	(* Internal method *)
	{attribute 'hide'}
	METHOD FB_init : BOOL
	VAR_INPUT
		(*  if TRUE, the retain variables are initialized (warm start / cold start) *)
		bInitRetains : BOOL;
		(*  if TRUE, the instance afterwards gets moved into the copy code (online change) *)
		bInCopyCode : BOOL;
	END_VAR
END_METHOD


	(* Internal method *)
	{attribute 'hide'}
	METHOD FB_exit : BOOL
	VAR_INPUT
		(*  if TRUE, the exit method is called for exiting an instance that is copied afterwards (online change). *)
		bInCopyCode : BOOL;
	END_VAR
END_METHOD


	(* Set the rotation angle in degrees [Â°]. *)
	METHOD SetAngle
	VAR_INPUT
		(* Rotation angle to set in degrees [Â°]. *)
		angle : LREAL;
	END_VAR
END_METHOD


	(* Set the components of this vector to '0.0'. *)
	METHOD SetZero
END_METHOD


	(* Set the components of this orientation. *)
	METHOD SetValues
	VAR_IN_OUT
		(* The position values to set. *)
 {attribute 'GUID' := '340DBC88-CE7F-36B9-693C-9000EEF35F3F'}
				orientation2D : Orientation2D;
	END_VAR
END_METHOD


	(* Get the direction of the local x-axis. *)
	METHOD GetDirectionX
	VAR_IN_OUT
		(* The local x-direction of this orientation. *)
 {attribute 'GUID' := 'FE5FBEA1-CCA0-3BC6-7207-1BBF2A5405AC'}
				localX : TangentXY;
	END_VAR
END_METHOD


	(* Get the direction of the local y-axis. *)
	METHOD GetDirectionY
	VAR_IN_OUT
		(* The local y-direction of this orientation. *)
 {attribute 'GUID' := 'FE5FBEA1-CCA0-3BC6-7207-1BBF2A5405AC'}
				localY : TangentXY;
	END_VAR
END_METHOD


	(* Invert this position. *)
	METHOD Invert
END_METHOD


	(* Multiply an orientation to this orientation. *)
	METHOD ConcatenateWith
	VAR_IN_OUT
		(* Orientation to concatenate with. *)
 {attribute 'GUID' := '340DBC88-CE7F-36B9-693C-9000EEF35F3F'}
				orientation2D : Orientation2D;
	END_VAR
END_METHOD


	(* Turn the orientation. *)
	METHOD TurnByC
	VAR_INPUT
		(* Rotation angle to turn by in degrees [Â°]. *)
		angle : LREAL;
	END_VAR
END_METHOD


	(* Rotate a PositionXY according to this orientation. *)
	METHOD Transform
	VAR_IN_OUT
		(* The orientation to multipy by. *)
 {attribute 'GUID' := '4E15B754-A8FD-31E0-757D-498AD44094D3'}
				positionXY : PositionXY;
	END_VAR
END_METHOD


	PROPERTY angle : LREAL
GET
END_GET
SET
END_SET
END_PROPERTY

END_FUNCTION_BLOCK

// POUs/Spatial/Functions/ConcatenateABC

	{attribute 'TcIecLibraryType'}
	{attribute 'external_name' := 'ConcatenateABC_GUID_C08B4073_E8F0_3BDB_7D4F_B552CCE66755'}
	(* Concatenate two instances of Orientation3D. *)
	FUNCTION ConcatenateABC : BOOL
	VAR_IN_OUT
		rotation0	:	Orientation3D;	(* 1st input orientation of the concatenation. *)
		rotation1	:	Orientation3D;	(* 2nd input orientation of the concatenation. *)
		concatenation	:	Orientation3D;	(* The concatenation of the two input instances. *)
	END_VAR

END_FUNCTION

// POUs/Spatial/Positions/Orientation3D

	{attribute 'c++_compatible'}
	{attribute 'external_name' := 'Orientation3D_GUID_50C17DBD_EDDF_3FDB_7A52_07B790BA3FF3'}
	{attribute 'TcIecLibraryType'}
	{attribute 'no_explicit_call' :='do not call this POU directly'}
	{attribute 'no_assign'}
	(* 3D orientation. All angles in degrees [Â°]. *)
	FUNCTION_BLOCK Orientation3D
	VAR
		(* Rotation around the 1st local axis in degrees [Â°]. *)
		p0 : LREAL;
		(* Rotation around 2nd local axis in degrees [Â°]. *)
		p1 : LREAL;
		(* Rotation around 3rd local axis in degrees [Â°]. *)
		p2 : LREAL;
		(* Defines the rotation order (rotate around local axes from left to right) *)
		 {attribute 'GUID' := 'BF8BCC1E-925E-4A57-801C-CC42AFDDA86D'}
		coordinates : E_RotationCoordinates := E_RotationCoordinates.CBA;
		 {attribute 'hide'}
		_reserved1 : ARRAY [1..84] OF USINT;
	END_VAR


	(* Internal method *)
	{attribute 'hide'}
	METHOD FB_init : BOOL
	VAR_INPUT
		(*  if TRUE, the retain variables are initialized (warm start / cold start) *)
		bInitRetains : BOOL;
		(*  if TRUE, the instance afterwards gets moved into the copy code (online change) *)
		bInCopyCode : BOOL;
	END_VAR
END_METHOD


	(* Internal method *)
	{attribute 'hide'}
	METHOD FB_exit : BOOL
	VAR_INPUT
		(*  if TRUE, the exit method is called for exiting an instance that is copied afterwards (online change). *)
		bInCopyCode : BOOL;
	END_VAR
END_METHOD


	(* Set the components of this vector to '0.0'. *)
	METHOD SetZero
END_METHOD


	(* Set the components of this position. *)
	METHOD SetValues
	VAR_IN_OUT
		(* The position values to set. *)
 {attribute 'GUID' := '50C17DBD-EDDF-3FDB-7A52-07B790BA3FF3'}
				orientation3D : Orientation3D;
	END_VAR
END_METHOD


	(* Set the coordinates of the orientation. *)
	METHOD SetValuesABC
	VAR_INPUT
		(* 1st rotation angle in degrees [Â°]. *)
		phi0 : LREAL;
		(* 2nd rotation angle in degrees [Â°]. *)
		phi1 : LREAL;
		(* 3rd rotation angle in degrees [Â°]. *)
		phi2 : LREAL;
	END_VAR
END_METHOD


	(* Set the coordinates of the orientation. *)
	METHOD SetValuesACB
	VAR_INPUT
		(* 1st rotation angle in degrees [Â°]. *)
		phi0 : LREAL;
		(* 2nd rotation angle in degrees [Â°]. *)
		phi1 : LREAL;
		(* 3rd rotation angle in degrees [Â°]. *)
		phi2 : LREAL;
	END_VAR
END_METHOD


	(* Set the coordinates of the orientation. *)
	METHOD SetValuesBCA
	VAR_INPUT
		(* 1st rotation angle in degrees [Â°]. *)
		phi0 : LREAL;
		(* 2nd rotation angle in degrees [Â°]. *)
		phi1 : LREAL;
		(* 3rd rotation angle in degrees [Â°]. *)
		phi2 : LREAL;
	END_VAR
END_METHOD


	(* Set the coordinates of the orientation. *)
	METHOD SetValuesBAC
	VAR_INPUT
		(* 1st rotation angle in degrees [Â°]. *)
		phi0 : LREAL;
		(* 2nd rotation angle in degrees [Â°]. *)
		phi1 : LREAL;
		(* 3rd rotation angle in degrees [Â°]. *)
		phi2 : LREAL;
	END_VAR
END_METHOD


	(* Set the coordinates of the orientation. *)
	METHOD SetValuesCAB
	VAR_INPUT
		(* 1st rotation angle in degrees [Â°]. *)
		phi0 : LREAL;
		(* 2nd rotation angle in degrees [Â°]. *)
		phi1 : LREAL;
		(* 3rd rotation angle in degrees [Â°]. *)
		phi2 : LREAL;
	END_VAR
END_METHOD


	(* Set the coordinates of the orientation. *)
	METHOD SetValuesCBA
	VAR_INPUT
		(* 1st rotation angle in degrees [Â°]. *)
		phi0 : LREAL;
		(* 2nd rotation angle in degrees [Â°]. *)
		phi1 : LREAL;
		(* 3rd rotation angle in degrees [Â°]. *)
		phi2 : LREAL;
	END_VAR
END_METHOD


	(* Set the coordinates of the orientation. *)
	METHOD SetValuesABA
	VAR_INPUT
		(* 1st rotation angle in degrees [Â°]. *)
		phi0 : LREAL;
		(* 2nd rotation angle in degrees [Â°]. *)
		phi1 : LREAL;
		(* 3rd rotation angle in degrees [Â°]. *)
		phi2 : LREAL;
	END_VAR
END_METHOD


	(* Set the coordinates of the orientation. *)
	METHOD SetValuesACA
	VAR_INPUT
		(* 1st rotation angle in degrees [Â°]. *)
		phi0 : LREAL;
		(* 2nd rotation angle in degrees [Â°]. *)
		phi1 : LREAL;
		(* 3rd rotation angle in degrees [Â°]. *)
		phi2 : LREAL;
	END_VAR
END_METHOD


	(* Set the coordinates of the orientation. *)
	METHOD SetValuesBCB
	VAR_INPUT
		(* 1st rotation angle in degrees [Â°]. *)
		phi0 : LREAL;
		(* 2nd rotation angle in degrees [Â°]. *)
		phi1 : LREAL;
		(* 3rd rotation angle in degrees [Â°]. *)
		phi2 : LREAL;
	END_VAR
END_METHOD


	(* Set the coordinates of the orientation. *)
	METHOD SetValuesBAB
	VAR_INPUT
		(* 1st rotation angle in degrees [Â°]. *)
		phi0 : LREAL;
		(* 2nd rotation angle in degrees [Â°]. *)
		phi1 : LREAL;
		(* 3rd rotation angle in degrees [Â°]. *)
		phi2 : LREAL;
	END_VAR
END_METHOD


	(* Set the coordinates of the orientation. *)
	METHOD SetValuesCAC
	VAR_INPUT
		(* 1st rotation angle in degrees [Â°]. *)
		phi0 : LREAL;
		(* 2nd rotation angle in degrees [Â°]. *)
		phi1 : LREAL;
		(* 3rd rotation angle in degrees [Â°]. *)
		phi2 : LREAL;
	END_VAR
END_METHOD


	(* Set the coordinates of the orientation. *)
	METHOD SetValuesCBC
	VAR_INPUT
		(* 1st rotation angle in degrees [Â°]. *)
		phi0 : LREAL;
		(* 2nd rotation angle in degrees [Â°]. *)
		phi1 : LREAL;
		(* 3rd rotation angle in degrees [Â°]. *)
		phi2 : LREAL;
	END_VAR
END_METHOD


	(* Get the direction of the local x-axis. *)
	METHOD GetDirectionX
	VAR_IN_OUT
		(* The local x-direction of this orientation. *)
 {attribute 'GUID' := '2D21607C-3841-350E-4823-AED297AC450B'}
				localX : Tangent3D;
	END_VAR
END_METHOD


	(* Get the direction of the local y-axis. *)
	METHOD GetDirectionY
	VAR_IN_OUT
		(* The local y-direction of this orientation. *)
 {attribute 'GUID' := '2D21607C-3841-350E-4823-AED297AC450B'}
				localY : Tangent3D;
	END_VAR
END_METHOD


	(* Get the direction of the local z-axis. *)
	METHOD GetDirectionZ
	VAR_IN_OUT
		(* The local z-direction of this orientation. *)
 {attribute 'GUID' := '2D21607C-3841-350E-4823-AED297AC450B'}
				localZ : Tangent3D;
	END_VAR
END_METHOD


	(* Invert this position. *)
	METHOD Invert
END_METHOD


	(* Multiply an orientation to this orientation. *)
	METHOD ConcatenateWith
	VAR_IN_OUT
		(* Orientation to concatenate with. *)
 {attribute 'GUID' := '50C17DBD-EDDF-3FDB-7A52-07B790BA3FF3'}
				orientation : Orientation3D;
	END_VAR
END_METHOD


	(* Rotate around an arbitrary local axis. The turn angle is given by the length of the axis. *)
	METHOD TurnBy
	VAR_IN_OUT
		(* The axis of rotation. Its length represents the angle of rotation in degrees [Â°]. *)
 {attribute 'GUID' := 'DF799042-141D-37B8-725F-419C4B15A84A'}
				axis : TangentABC;
	END_VAR
END_METHOD


	(* Rotation around the local x-axis. *)
	METHOD TurnByA
	VAR_INPUT
		(* The angle to rotate by in degrees [Â°]. *)
		da : LREAL;
	END_VAR
END_METHOD


	(* Rotation around the local y-axis. *)
	METHOD TurnByB
	VAR_INPUT
		(* The angle to rotate by in degrees [Â°]. *)
		db : LREAL;
	END_VAR
END_METHOD


	(* Rotation around the local z-axis. *)
	METHOD TurnByC
	VAR_INPUT
		(* The angle to rotate by in degrees [Â°]. *)
		dc : LREAL;
	END_VAR
END_METHOD


	(* Rotate a Position3D according to this orientation. *)
	METHOD Transform
	VAR_IN_OUT
		(* Position to transform. *)
 {attribute 'GUID' := 'F25F0046-C763-3F00-5FBE-159880852C99'}
				position3D : Position3D;
	END_VAR
END_METHOD


	PROPERTY phi0 : LREAL
GET
END_GET
SET
END_SET
END_PROPERTY


	PROPERTY phi1 : LREAL
GET
END_GET
SET
END_SET
END_PROPERTY


	PROPERTY phi2 : LREAL
GET
END_GET
SET
END_SET
END_PROPERTY


	PROPERTY convention : E_RotationCoordinates
GET
END_GET
SET
END_SET
END_PROPERTY

END_FUNCTION_BLOCK

// POUs/Spatial/Functions/ConcatenateXYC

	{attribute 'TcIecLibraryType'}
	{attribute 'external_name' := 'ConcatenateXYC_GUID_E714162A_B2D1_3B7D_7D74_ACE9FDB339B0'}
	(* Concatenate two instances of PositionXYC. *)
	FUNCTION ConcatenateXYC : BOOL
	VAR_IN_OUT
		position0	:	PositionXYC;	(* 1st input position of the concatenation. *)
		position1	:	PositionXYC;	(* 2nd input position of the concatenation. *)
		concatenation	:	PositionXYC;	(* The concatenation of the two input instances. *)
	END_VAR

END_FUNCTION

// POUs/Spatial/Functions/Concatenate6D

	{attribute 'TcIecLibraryType'}
	{attribute 'external_name' := 'Concatenate6D_GUID_117C0CA0_BCAB_3F0B_4FE1_4D251F2AE781'}
	(* Concatenate two instances of PositionSE3. *)
	FUNCTION Concatenate6D : BOOL
	VAR_IN_OUT
		position0	:	PositionSE3;	(* 1st input position of the concatenation. *)
		position1	:	PositionSE3;	(* 2nd input position of the concatenation. *)
		concatenation	:	PositionXYC;	(* The concatenation of the two input instances. *)
	END_VAR

END_FUNCTION

// POUs/Spatial/Functions/AddXY

	{attribute 'TcIecLibraryType'}
	{attribute 'external_name' := 'AddXY_GUID_4211BB55_4701_355E_49B7_FBB5A6A56D0F'}
	(* Add two instances of TangentXY. *)
	FUNCTION AddXY : BOOL
	VAR_IN_OUT
		tangent0	:	TangentXY;	(* 1st input tangent vector. *)
		tangent1	:	TangentXY;	(* 2nd input tangent vector. *)
		sumTangent	:	TangentXY;	(* Sum of the two tangent vectors. *)
	END_VAR

END_FUNCTION

// POUs/Spatial/Functions/SubtractXY

	{attribute 'TcIecLibraryType'}
	{attribute 'external_name' := 'SubtractXY_GUID_93ADB8A4_4C15_3784_788B_007580BC0FF8'}
	(* Subtract two instances of TangentXY. *)
	FUNCTION SubtractXY : BOOL
	VAR_IN_OUT
		tangent0	:	TangentXY;	(* 1st input tangent vector. *)
		tangent1	:	TangentXY;	(* 2nd input tangent vector. *)
		difference	:	TangentXY;	(* Difference of the two tangent vectors. *)
	END_VAR

END_FUNCTION

// POUs/Spatial/Functions/MultiplyXY

	{attribute 'TcIecLibraryType'}
	{attribute 'external_name' := 'MultiplyXY_GUID_5D064EB0_5BE0_3721_7F02_812C9FF897A8'}
	(* Multiply a TangentXY by a scalar and return the result. *)
	FUNCTION MultiplyXY : BOOL
	VAR_IN_OUT
		tangent	:	TangentXY;	(* Tangent vector to multiply. *)
	END_VAR
	VAR_INPUT
		scalar	:	LREAL;	(* Scalar value to multiply with. *)
	END_VAR
	VAR_IN_OUT
		scaled	:	TangentXY;	(* Scaled input tangent vector. *)
	END_VAR

END_FUNCTION

// POUs/Spatial/Functions/ScalarXY

	{attribute 'TcIecLibraryType'}
	{attribute 'external_name' := 'ScalarXY_GUID_4B1B8ECC_B5D0_31F8_77A8_B617B525F46F'}
	(* Compute the scalar product of two instance of TangentXY. *)
	FUNCTION ScalarXY : LREAL
	VAR_IN_OUT
		tangent0	:	TangentXY;	(* 1st input tangent vector. *)
		tangent1	:	TangentXY;	(* 2nd input tangent vector. *)
	END_VAR

END_FUNCTION

// POUs/Spatial/Functions/Add3D

	{attribute 'TcIecLibraryType'}
	{attribute 'external_name' := 'Add3D_GUID_81D10FB6_FC18_39A3_5098_92A645D8B8D4'}
	(* Add two instances of Tangent3D. *)
	FUNCTION Add3D : BOOL
	VAR_IN_OUT
		tangent0	:	Tangent3D;	(* 1st input tangent vector. *)
		tangent1	:	Tangent3D;	(* 2nd input tangent vector. *)
		sumTangent	:	Tangent3D;	(* Sum of the two tangent vectors. *)
	END_VAR

END_FUNCTION

// POUs/Spatial/Functions/Subtract3D

	{attribute 'TcIecLibraryType'}
	{attribute 'external_name' := 'Subtract3D_GUID_9C77A7E2_4702_3C0D_7E52_C6A53DEA5206'}
	(* Subtract two instances of Tangent3D. *)
	FUNCTION Subtract3D : BOOL
	VAR_IN_OUT
		tangent0	:	Tangent3D;	(* 1st input tangent vector. *)
		tangent1	:	Tangent3D;	(* 2nd input tangent vector. *)
		difference	:	Tangent3D;	(* Difference of the two tangent vectors. *)
	END_VAR

END_FUNCTION

// POUs/Spatial/Functions/Multiply3D

	{attribute 'TcIecLibraryType'}
	{attribute 'external_name' := 'Multiply3D_GUID_E0D20371_4D68_3851_702C_6480A326A604'}
	(* Multiply a Tangent3D by a scalar. *)
	FUNCTION Multiply3D : BOOL
	VAR_IN_OUT
		tangent	:	Tangent3D;	(* Tangent vector to multiply. *)
	END_VAR
	VAR_INPUT
		scalar	:	LREAL;	(* Scalar value to multiply with. *)
	END_VAR
	VAR_IN_OUT
		scaled	:	Tangent3D;	(* Scaled input tangent vector. *)
	END_VAR

END_FUNCTION

// POUs/Spatial/Functions/Scalar3D

	{attribute 'TcIecLibraryType'}
	{attribute 'external_name' := 'Scalar3D_GUID_1532A384_100A_3B48_6D65_E3904A6F9DEC'}
	(* Compute the scalar product of two instances of Tangent3D. *)
	FUNCTION Scalar3D : LREAL
	VAR_IN_OUT
		tangent0	:	Tangent3D;	(* 1st input tangent vector. *)
		tangent1	:	Tangent3D;	(* 2nd input tangent vector. *)
	END_VAR

END_FUNCTION

// POUs/Spatial/Functions/Cross3D

	{attribute 'TcIecLibraryType'}
	{attribute 'external_name' := 'Cross3D_GUID_C01A5103_5AD1_3885_5546_AB884404E9D1'}
	(* Compute the cross product of two instances of Tangent3D. *)
	FUNCTION Cross3D : BOOL
	VAR_IN_OUT
		tangent0	:	Tangent3D;	(* 1st input tangent vector. *)
		tangent1	:	Tangent3D;	(* 2nd input tangent vector. *)
		crossProduct	:	Tangent3D;	(* The resulting cross product. *)
	END_VAR

END_FUNCTION

// POUs/Spatial/Functions/AddABC

	{attribute 'TcIecLibraryType'}
	{attribute 'external_name' := 'AddABC_GUID_101C95D8_FA86_369B_4FDE_199CF7ED8C7A'}
	(* Add two instances of TangentABC. *)
	FUNCTION AddABC : BOOL
	VAR_IN_OUT
		tangent0	:	TangentABC;	(* 1st input tangent vector. *)
		tangent1	:	TangentABC;	(* 2nd input tangent vector. *)
		sumTangent	:	TangentABC;	(* Sum of the two tangent vectors. *)
	END_VAR

END_FUNCTION

// POUs/Spatial/Functions/SubtractABC

	{attribute 'TcIecLibraryType'}
	{attribute 'external_name' := 'SubtractABC_GUID_ADA30DD9_D160_3448_7A2B_2846F825BFFF'}
	(* Subtract two instances of TangentABC. *)
	FUNCTION SubtractABC : BOOL
	VAR_IN_OUT
		tangent0	:	TangentABC;	(* 1st input tangent vector. *)
		tangent1	:	TangentABC;	(* 2nd input tangent vector. *)
		difference	:	TangentABC;	(* Difference of the two tangent vectors. *)
	END_VAR

END_FUNCTION

// POUs/Spatial/Functions/MultiplyABC

	{attribute 'TcIecLibraryType'}
	{attribute 'external_name' := 'MultiplyABC_GUID_6DB10CD6_2FBE_3B0D_6DB1_2A11ABD146D1'}
	(* Multiply a TangentABC by a scalar. *)
	FUNCTION MultiplyABC : BOOL
	VAR_IN_OUT
		tangent	:	TangentABC;	(* Tangent vector to multiply. *)
	END_VAR
	VAR_INPUT
		scalar	:	LREAL;	(* Scalar value to multiply with. *)
	END_VAR
	VAR_IN_OUT
		scaled	:	TangentABC;	(* Scaled input tangent vector. *)
	END_VAR

END_FUNCTION

// POUs/Spatial/Functions/AddXYC

	{attribute 'TcIecLibraryType'}
	{attribute 'external_name' := 'AddXYC_GUID_BD7038A3_BE3D_3097_7032_654AEC111158'}
	(* Add two instances of TangentXYC. *)
	FUNCTION AddXYC : BOOL
	VAR_IN_OUT
		tangent0	:	TangentXYC;	(* 1st input tangent vector. *)
		tangent1	:	TangentXYC;	(* 2nd input tangent vector. *)
		sumTangent	:	TangentXYC;	(* Sum of the two tangent vectors. *)
	END_VAR

END_FUNCTION

// POUs/Spatial/Functions/SubtractXYC

	{attribute 'TcIecLibraryType'}
	{attribute 'external_name' := 'SubtractXYC_GUID_7E8D6E3C_EDF3_3ECD_4F27_E6795E207B1F'}
	(* Subtract two instances of TangentXYC. *)
	FUNCTION SubtractXYC : BOOL
	VAR_IN_OUT
		tangent0	:	TangentXYC;	(* 1st input tangent vector. *)
		tangent1	:	TangentXYC;	(* 2nd input tangent vector. *)
		difference	:	TangentXYC;	(* Difference of the two tangent vectors. *)
	END_VAR

END_FUNCTION

// POUs/Spatial/Functions/MultiplyXYC

	{attribute 'TcIecLibraryType'}
	{attribute 'external_name' := 'MultiplyXYC_GUID_C857FA2E_ED30_35BE_4A13_1DEC370C7D45'}
	(* Multiply a TangentXYC by a scalar. *)
	FUNCTION MultiplyXYC : BOOL
	VAR_IN_OUT
		tangent	:	TangentXYC;	(* Tangent vector to multiply. *)
	END_VAR
	VAR_INPUT
		scalar	:	LREAL;	(* Scalar value to multiply with. *)
	END_VAR
	VAR_IN_OUT
		scaled	:	TangentXYC;	(* Scaled input tangent vector. *)
	END_VAR

END_FUNCTION

// POUs/Spatial/Functions/Add6D

	{attribute 'TcIecLibraryType'}
	{attribute 'external_name' := 'Add6D_GUID_A8706E90_BB9B_3CBB_7DD4_65F4D3621CA7'}
	(* Add two instances of Tangent6D. *)
	FUNCTION Add6D : BOOL
	VAR_IN_OUT
		tangent0	:	Tangent6D;	(* 1st input tangent vector. *)
		tangent1	:	Tangent6D;	(* 2nd input tangent vector. *)
		sumTangent	:	Tangent6D;	(* Sum of the two tangent vectors. *)
	END_VAR

END_FUNCTION

// POUs/Spatial/Functions/Subtract6D

	{attribute 'TcIecLibraryType'}
	{attribute 'external_name' := 'Subtract6D_GUID_5DE3145A_A69E_3354_58A7_9855101F40EC'}
	(* Subtract two instances of Tangent6D. *)
	FUNCTION Subtract6D : BOOL
	VAR_IN_OUT
		tangent0	:	Tangent6D;	(* 1st input tangent vector. *)
		tangent1	:	Tangent6D;	(* 2nd input tangent vector. *)
		difference	:	Tangent6D;	(* Difference of the two tangent vectors. *)
	END_VAR

END_FUNCTION

// POUs/Spatial/Functions/Multiply6D

	{attribute 'TcIecLibraryType'}
	{attribute 'external_name' := 'Multiply6D_GUID_49BE7CCB_C420_30B9_422A_6CCBC76FF2E8'}
	(* Multiply a Tangent6D by a scalar. *)
	FUNCTION Multiply6D : BOOL
	VAR_IN_OUT
		tangent	:	Tangent6D;	(* Tangent vector to multiply. *)
	END_VAR
	VAR_INPUT
		scalar	:	LREAL;	(* Scalar value to multiply with. *)
	END_VAR
	VAR_IN_OUT
		scaled	:	Tangent6D;	(* Scaled input tangent vector. *)
	END_VAR

END_FUNCTION

// POUs/Spatial/Functions/ConvertToCartesian2D

	{attribute 'TcIecLibraryType'}
	{attribute 'external_name' := 'ConvertToCartesian2D_GUID_C5072885_CC2B_39CB_7DF2_74FA29D8F10B'}
	(* Convert local XYC-dynamic properties to global XY ones. *)
	FUNCTION ConvertToCartesian2D : BOOL
	VAR_IN_OUT
		position	:	PositionXYC;	(* The position hosting the local dynamic state. *)
		velocity	:	TangentXYC;	(* The local velocity vector. *)
		acceleration	:	TangentXYC;	(* The local acceleration vector. *)
		velocity_XY	:	TangentXY;	(* The resulting global Cartesian velocity. *)
		acceleration_XY	:	TangentXY;	(* The resulting global Cartesian acceleration. *)
	END_VAR

END_FUNCTION

// POUs/Spatial/Setpoints/SetpointR1

	{attribute 'c++_compatible'}
	{attribute 'external_name' := 'SetpointR1_GUID_941F0815_CD7F_3A56_4D2C_59489EF46EE2'}
	{attribute 'TcIecLibraryType'}
	{attribute 'no_explicit_call' :='do not call this POU directly'}
	{attribute 'no_assign_warning'}
	(* 1D setpoint. *)
	FUNCTION_BLOCK SetpointR1
	VAR
		(* Position component of the setpoint. *)
		ds : LREAL;
		(* Velocity component of the setpoint. *)
		dv : LREAL;
		(* Acceleration component of the setpoint. *)
		da : LREAL;
		(* Jerk component of the setpoint. *)
		dj : LREAL;
	END_VAR


	(* Internal method *)
	{attribute 'hide'}
	METHOD FB_init : BOOL
	VAR_INPUT
		(*  if TRUE, the retain variables are initialized (warm start / cold start) *)
		bInitRetains : BOOL;
		(*  if TRUE, the instance afterwards gets moved into the copy code (online change) *)
		bInCopyCode : BOOL;
	END_VAR
END_METHOD


	(* Internal method *)
	{attribute 'hide'}
	METHOD FB_reinit : BOOL
END_METHOD


	(* Internal method *)
	{attribute 'hide'}
	METHOD FB_exit : BOOL
	VAR_INPUT
		(*  if TRUE, the exit method is called for exiting an instance that is copied afterwards (online change). *)
		bInCopyCode : BOOL;
	END_VAR
END_METHOD


	(* Set this setpoint to zero. *)
	METHOD SetZero
END_METHOD


	(* Set the values of this coordinate. *)
	METHOD SetValuesSVAJ
	VAR_INPUT
		(* the position value to set. *)
		_s : LREAL;
		(* the velocity value to set. *)
		v : LREAL;
		(* the acceleration value to set. *)
		a : LREAL;
		(* the jerk value to set. *)
		j : LREAL;
	END_VAR
END_METHOD


	PROPERTY _s : LREAL
GET
END_GET
SET
END_SET
END_PROPERTY


	PROPERTY v : LREAL
GET
END_GET
SET
END_SET
END_PROPERTY


	PROPERTY a : LREAL
GET
END_GET
SET
END_SET
END_PROPERTY


	PROPERTY j : LREAL
GET
END_GET
SET
END_SET
END_PROPERTY

END_FUNCTION_BLOCK

// POUs/Spatial/Setpoints/SetpointSE3

	{attribute 'c++_compatible'}
	{attribute 'external_name' := 'SetpointSE3_GUID_0090A85D_3232_323F_6DC4_D19BCED5289D'}
	{attribute 'TcIecLibraryType'}
	{attribute 'no_explicit_call' :='do not call this POU directly'}
	{attribute 'no_assign_warning'}
	(* SE3 setpoint. *)
	FUNCTION_BLOCK SetpointSE3 EXTENDS IPlcGeometry3D


	(* Internal method *)
	{attribute 'hide'}
	METHOD FB_init : BOOL
	VAR_INPUT
		(*  if TRUE, the retain variables are initialized (warm start / cold start) *)
		bInitRetains : BOOL;
		(*  if TRUE, the instance afterwards gets moved into the copy code (online change) *)
		bInCopyCode : BOOL;
	END_VAR
END_METHOD


	(* Internal method *)
	{attribute 'hide'}
	METHOD FB_exit : BOOL
	VAR_INPUT
		(*  if TRUE, the exit method is called for exiting an instance that is copied afterwards (online change). *)
		bInCopyCode : BOOL;
	END_VAR
END_METHOD


	(* Set this setpoint to be the identity. *)
	METHOD SetIdentity
END_METHOD


	(* Set the values of this setpoint. *)
	METHOD SetValues
	VAR_IN_OUT
		(* The setpoint to copy. *)
 {attribute 'GUID' := '0090A85D-3232-323F-6DC4-D19BCED5289D'}
				setpoint : SetpointSE3;
	END_VAR
END_METHOD


	(* Set the cartesian values of this setpoint. *)
	METHOD SetValuesXYZ
	VAR_IN_OUT
		(* The x-setpoint to set. *)
 {attribute 'GUID' := '941F0815-CD7F-3A56-4D2C-59489EF46EE2'}
				setpointX : SetpointR1;
		(* The y-setpoint to set. *)
 {attribute 'GUID' := '941F0815-CD7F-3A56-4D2C-59489EF46EE2'}
				setpointY : SetpointR1;
		(* The z-setpoint to set. *)
 {attribute 'GUID' := '941F0815-CD7F-3A56-4D2C-59489EF46EE2'}
				setpointZ : SetpointR1;
	END_VAR
END_METHOD


	(* Set the angular values of this setpoint. *)
	METHOD SetValuesCBA
	VAR_IN_OUT
		(* The c-setpoint to set. *)
 {attribute 'GUID' := '941F0815-CD7F-3A56-4D2C-59489EF46EE2'}
				setpointC : SetpointR1;
		(* The b-setpoint to set. *)
 {attribute 'GUID' := '941F0815-CD7F-3A56-4D2C-59489EF46EE2'}
				setpointB : SetpointR1;
		(* The a-setpoint to set. *)
 {attribute 'GUID' := '941F0815-CD7F-3A56-4D2C-59489EF46EE2'}
				setpointA : SetpointR1;
	END_VAR
END_METHOD


	(* Get the direction of the local x-axis. *)
	METHOD GetDirectionX
	VAR_IN_OUT
		(* The local x-direction of this orientation. *)
 {attribute 'GUID' := '2D21607C-3841-350E-4823-AED297AC450B'}
				localX : Tangent3D;
	END_VAR
END_METHOD


	(* Get the direction of the local y-axis. *)
	METHOD GetDirectionY
	VAR_IN_OUT
		(* The local y-direction of this orientation. *)
 {attribute 'GUID' := '2D21607C-3841-350E-4823-AED297AC450B'}
				localY : Tangent3D;
	END_VAR
END_METHOD


	(* Get the direction of the local z-axis. *)
	METHOD GetDirectionZ
	VAR_IN_OUT
		(* The local z-direction of this orientation. *)
 {attribute 'GUID' := '2D21607C-3841-350E-4823-AED297AC450B'}
				localZ : Tangent3D;
	END_VAR
END_METHOD


	(* Get the linear Cartesian position components. *)
	METHOD GetPosition_Cartesian
	VAR_IN_OUT
		(* The output position. *)
 {attribute 'GUID' := 'F25F0046-C763-3F00-5FBE-159880852C99'}
				position : Position3D;
	END_VAR
END_METHOD


	(* Get the linear Cartesian velocity components. *)
	METHOD GetVelocity_Cartesian
	VAR_IN_OUT
		(* The output tangent. *)
 {attribute 'GUID' := '2D21607C-3841-350E-4823-AED297AC450B'}
				tangent : Tangent3D;
	END_VAR
END_METHOD


	(* Get the linear Cartesian acceleration components. *)
	METHOD GetAcceleration_Cartesian
	VAR_IN_OUT
		(* The output tangent. *)
 {attribute 'GUID' := '2D21607C-3841-350E-4823-AED297AC450B'}
				tangent : Tangent3D;
	END_VAR
END_METHOD


	(* Get the linear Cartesian jerk components. *)
	METHOD GetJerk_Cartesian
	VAR_IN_OUT
		(* The output tangent. *)
 {attribute 'GUID' := '2D21607C-3841-350E-4823-AED297AC450B'}
				tangent : Tangent3D;
	END_VAR
END_METHOD


	(* Concatenate this setpoint with a second one up to a specific order. *)
	METHOD ConcatenateWith
	VAR_IN_OUT
		(* The setpoint to concatenate. *)
 {attribute 'GUID' := '0090A85D-3232-323F-6DC4-D19BCED5289D'}
				setpoint : SetpointSE3;
	END_VAR
	VAR_INPUT
		(*  The order up to which to compute. *)
		order : UDINT;
	END_VAR
END_METHOD


	PROPERTY x : LREAL
GET
END_GET
SET
END_SET
END_PROPERTY


	PROPERTY y : LREAL
GET
END_GET
SET
END_SET
END_PROPERTY


	PROPERTY z : LREAL
GET
END_GET
SET
END_SET
END_PROPERTY


	PROPERTY phi0 : LREAL
GET
END_GET
SET
END_SET
END_PROPERTY


	PROPERTY phi1 : LREAL
GET
END_GET
SET
END_SET
END_PROPERTY


	PROPERTY phi2 : LREAL
GET
END_GET
SET
END_SET
END_PROPERTY


	PROPERTY Convention : E_RotationCoordinates
GET
END_GET
SET
END_SET
END_PROPERTY

END_FUNCTION_BLOCK

// POUs/Spatial/Inertias/InertiaSE3

	{attribute 'c++_compatible'}
	{attribute 'external_name' := 'InertiaSE3_GUID_98C1A030_EB37_3B8D_427A_BFDCFF6C5618'}
	{attribute 'TcIecLibraryType'}
	{attribute 'no_explicit_call' :='do not call this POU directly'}
	{attribute 'no_assign'}
	(* Inertia tensor containing angular and linear inertia. *)
	FUNCTION_BLOCK InertiaSE3
	VAR
		(* Mass of the inertia. *)
		m : LREAL;
		(* x-component of the center of mass. *)
		CenterX : LREAL;
		(* y-component of the center of mass. *)
		CenterY : LREAL;
		(* z-component of the center of mass. *)
		CenterZ : LREAL;
		 {attribute 'hide'}
		_reserved1 : ARRAY [1..80] OF USINT;
	END_VAR


	(* Internal method *)
	{attribute 'hide'}
	METHOD FB_init : BOOL
	VAR_INPUT
		(*  if TRUE, the retain variables are initialized (warm start / cold start) *)
		bInitRetains : BOOL;
		(*  if TRUE, the instance afterwards gets moved into the copy code (online change) *)
		bInCopyCode : BOOL;
	END_VAR
END_METHOD


	(* Internal method *)
	{attribute 'hide'}
	METHOD FB_exit : BOOL
	VAR_INPUT
		(*  if TRUE, the exit method is called for exiting an instance that is copied afterwards (online change). *)
		bInCopyCode : BOOL;
	END_VAR
END_METHOD


	(* Add a 2nd inertia tensor to this one. *)
	METHOD AddBy
	VAR_IN_OUT
		(* The inertia tensor to add. *)
 {attribute 'GUID' := '98C1A030-EB37-3B8D-427A-BFDCFF6C5618'}
				shift : InertiaSE3;
	END_VAR
END_METHOD


	(* Set the values to that of a point. *)
	METHOD SetValues_Point
	VAR_INPUT
		(* The mass of the point. *)
		mass : LREAL;
		(* The x-position of the point. *)
		x : LREAL;
		(* The y-position of the point. *)
		y : LREAL;
		(* The z-position of the point. *)
		z : LREAL;
	END_VAR
END_METHOD


	(* Set the values to that of a sphere. *)
	METHOD SetValues_Sphere
	VAR_INPUT
		(* The mass of the sphere. *)
		mass : LREAL;
		(* The radius of the sphere. *)
		radius : LREAL;
	END_VAR
END_METHOD


	(* Set the values to that of a cylinder. *)
	METHOD SetValues_Cylinder
	VAR_INPUT
		(* The mass of the cylinder. *)
		mass : LREAL;
		(* The radius of the cylinder. *)
		radius : LREAL;
		(* The height of the cylinder. *)
		height : LREAL;
	END_VAR
END_METHOD


	(* Set the values to that of a cuboid. *)
	METHOD SetValues_Cuboid
	VAR_INPUT
		(* The mass of the cuboid. *)
		mass : LREAL;
		(* The x-length of the cuboid. *)
		dx : LREAL;
		(* The y-length of the cuboid. *)
		dy : LREAL;
		(* The z-length of the cuboid. *)
		dz : LREAL;
	END_VAR
END_METHOD


	(* Transform this inertia by a displacement. *)
	METHOD Transform
	VAR_IN_OUT
		(* The displacement to apply. *)
 {attribute 'GUID' := 'D2337217-563D-354C-4349-0B99B7C3F40C'}
				displacement : PositionSE3;
	END_VAR
END_METHOD


	(* Translate this inertia by a translation. *)
	METHOD Translate
	VAR_IN_OUT
		(* The translation to apply. *)
 {attribute 'GUID' := '2D21607C-3841-350E-4823-AED297AC450B'}
				displacement : Tangent3D;
	END_VAR
END_METHOD


	PROPERTY mass : LREAL
GET
END_GET
SET
END_SET
END_PROPERTY


	PROPERTY x : LREAL
GET
END_GET
SET
END_SET
END_PROPERTY


	PROPERTY y : LREAL
GET
END_GET
SET
END_SET
END_PROPERTY


	PROPERTY z : LREAL
GET
END_GET
SET
END_SET
END_PROPERTY


	PROPERTY xx : LREAL
GET
END_GET
SET
END_SET
END_PROPERTY


	PROPERTY yy : LREAL
GET
END_GET
SET
END_SET
END_PROPERTY


	PROPERTY zz : LREAL
GET
END_GET
SET
END_SET
END_PROPERTY


	PROPERTY xy : LREAL
GET
END_GET
SET
END_SET
END_PROPERTY


	PROPERTY yz : LREAL
GET
END_GET
SET
END_SET
END_PROPERTY


	PROPERTY zx : LREAL
GET
END_GET
SET
END_SET
END_PROPERTY

END_FUNCTION_BLOCK

// POUs/Shapes/Geometry2D/Container2D

	{attribute 'c++_compatible'}
	{attribute 'external_name' := 'Container2D_GUID_E9BC710F_698E_36D4_4508_020D28DA2F7D'}
	{attribute 'TcIecLibraryType'}
	{attribute 'no_explicit_call' :='do not call this POU directly'}
	{attribute 'no_assign'}
	FUNCTION_BLOCK Container2D EXTENDS Geometry2D


	(* Internal method *)
	METHOD FB_init : BOOL
	VAR_INPUT
		(*  if TRUE, the retain variables are initialized (warm start / cold start) *)
		bInitRetains : BOOL;
		(*  if TRUE, the instance afterwards gets moved into the copy code (online change) *)
		bInCopyCode : BOOL;
	END_VAR
END_METHOD


	(* Internal method *)
	{attribute 'hide'}
	METHOD FB_exit : BOOL
	VAR_INPUT
		(*  if TRUE, the exit method is called for exiting an instance that is copied afterwards (online change). *)
		bInCopyCode : BOOL;
	END_VAR
END_METHOD


	(* Add a geometry to the container. *)
	METHOD AddElement : UDINT
	VAR_IN_OUT
		(* The geometry to add. *)
 {attribute 'GUID' := '75DBC672-BA4B-3F92-667E-BA753274B090'}
				inputObject : Geometry2D;
	END_VAR
END_METHOD


	(* Remove a specified geometry from the container. *)
	METHOD RemoveElement
	VAR_INPUT
		(* ID of the geometry to remove. *)
		id : UDINT;
	END_VAR
END_METHOD


	(* Remove all geometries from the container. *)
	METHOD Clear
END_METHOD


	(* Get the number of geometry elements in container. *)
	METHOD GetCount : UDINT
END_METHOD


	(* Get the combined boundary of all hosted 2D-geometries. *)
	METHOD GetBoundary
	VAR_IN_OUT
		(* The combined boundary.. *)
 {attribute 'GUID' := 'E9BC710F-698E-36D4-4508-020D28DA2F7D'}
				boundary : Container2D;
	END_VAR
END_METHOD

END_FUNCTION_BLOCK

// POUs/Shapes/Geometry2D/Extrude2D

	{attribute 'c++_compatible'}
	{attribute 'external_name' := 'Extrude2D_GUID_7FDEF7A4_92FB_356D_4B02_9EF0BC3A7BB4'}
	{attribute 'TcIecLibraryType'}
	{attribute 'no_explicit_call' :='do not call this POU directly'}
	{attribute 'no_assign'}
	FUNCTION_BLOCK Extrude2D EXTENDS Geometry2D


	(* Internal method *)
	METHOD FB_init : BOOL
	VAR_INPUT
		(*  if TRUE, the retain variables are initialized (warm start / cold start) *)
		bInitRetains : BOOL;
		(*  if TRUE, the instance afterwards gets moved into the copy code (online change) *)
		bInCopyCode : BOOL;
	END_VAR
END_METHOD


	(* Internal method *)
	{attribute 'hide'}
	METHOD FB_exit : BOOL
	VAR_INPUT
		(*  if TRUE, the exit method is called for exiting an instance that is copied afterwards (online change). *)
		bInCopyCode : BOOL;
	END_VAR
END_METHOD


	(* Define the extrusion geometry by a path and the corners to extrude. *)
	METHOD ExtrudeAlong
	VAR_IN_OUT
		(* The path to extrude along. *)
 {attribute 'GUID' := 'DCABE934-067B-358F-63E2-89B9B6F161E3'}
				path : PathXYC;
	END_VAR
	VAR_INPUT
		(* 1st distance from the path to extrude. *)
		dy0 : LREAL;
		(* 2nd distance from the path to extrude. *)
		dy1 : LREAL;
		(* Number of steps to employ along the path. *)
		extrusionSteps : UDINT;
	END_VAR
END_METHOD


	(* Check whether this extrusion geometry is valid. *)
	METHOD IsValid : BOOL
END_METHOD

END_FUNCTION_BLOCK

// POUs/Paths/Components/PathXYC

	{attribute 'c++_compatible'}
	{attribute 'external_name' := 'PathXYC_GUID_DCABE934_067B_358F_63E2_89B9B6F161E3'}
	{attribute 'TcIecLibraryType'}
	{attribute 'no_explicit_call' :='do not call this POU directly'}
	{attribute 'no_assign'}
	(* A path in the xy-plane with an additional orientation at every path position. *)
	FUNCTION_BLOCK PathXYC EXTENDS IPlcPath2D


	(* Internal method *)
	{attribute 'hide'}
	METHOD FB_init : BOOL
	VAR_INPUT
		(*  if TRUE, the retain variables are initialized (warm start / cold start) *)
		bInitRetains : BOOL;
		(*  if TRUE, the instance afterwards gets moved into the copy code (online change) *)
		bInCopyCode : BOOL;
	END_VAR
END_METHOD


	(* Internal method *)
	{attribute 'hide'}
	METHOD FB_exit : BOOL
	VAR_INPUT
		(*  if TRUE, the exit method is called for exiting an instance that is copied afterwards (online change). *)
		bInCopyCode : BOOL;
	END_VAR
END_METHOD


	(* Append a smooth transition from the current end of the path
				    to the specified position. *)
	METHOD AppendPosition
	VAR_IN_OUT
		(* The position to append. *)
 {attribute 'GUID' := 'CB2F0EE9-C51F-39A6-6052-0A7E5AD17161'}
				position : PositionXYC;
	END_VAR
END_METHOD


	(* Append a smooth transition from the current end of the path
				    to the specified position. *)
	METHOD AppendPositionXYC
	VAR_INPUT
		(* x-component of the position to append. *)
		x : LREAL;
		(* y-component of the position to append. *)
		y : LREAL;
		(* c-component of the position to append in degrees [Â°]. *)
		c : LREAL;
	END_VAR
END_METHOD


	(* Append a line to this path. *)
	METHOD AppendLine
	VAR_IN_OUT
		(* Start position of the line. *)
 {attribute 'GUID' := 'CB2F0EE9-C51F-39A6-6052-0A7E5AD17161'}
				startPos : PositionXYC;
		(* End position of the line. *)
 {attribute 'GUID' := 'CB2F0EE9-C51F-39A6-6052-0A7E5AD17161'}
				endPos : PositionXYC;
	END_VAR
END_METHOD


	(* Append a circle to this path. *)
	METHOD AppendCircle
	VAR_IN_OUT
		(* Start position of the circle. *)
 {attribute 'GUID' := 'CB2F0EE9-C51F-39A6-6052-0A7E5AD17161'}
				startPos : PositionXYC;
		(* End position of the circle. *)
 {attribute 'GUID' := 'CB2F0EE9-C51F-39A6-6052-0A7E5AD17161'}
				endPos : PositionXYC;
		(* Center of the circle. *)
 {attribute 'GUID' := '4E15B754-A8FD-31E0-757D-498AD44094D3'}
				center : PositionXY;
	END_VAR
	VAR_INPUT
		(* Set whether the circle runs clockwise or counter-clockwise. *)
		clockwise : BOOL;
	END_VAR
END_METHOD


	(* Appends a smooth transition from the end of this path
				      to the start of the other path, locking further changes of this path. *)
	METHOD EndAtPath
	VAR_IN_OUT
		(* The other path. *)
 {attribute 'GUID' := 'DCABE934-067B-358F-63E2-89B9B6F161E3'}
				path : PathXYC;
	END_VAR
END_METHOD


	(* Appends a smooth transition from the start of this path
				      to the end of the other path, locking further changes of the other path. *)
	METHOD StartFromPath
	VAR_IN_OUT
		(* The other path. *)
 {attribute 'GUID' := 'DCABE934-067B-358F-63E2-89B9B6F161E3'}
				path : PathXYC;
	END_VAR
END_METHOD


	(* Connect start and end position.
				      A smooth transition is added as long as start and end positin are not identical.
				      This operation finalizes this path definition and locks it against further modifications. *)
	METHOD CloseLoop
END_METHOD


	(* Empty all current path definitions and reset the path back to an empty state. *)
	METHOD Clear
END_METHOD


	(* Get the start position of the path. *)
	METHOD GetStartPosition
	VAR_IN_OUT
		(* The current start position of the path. *)
 {attribute 'GUID' := 'CB2F0EE9-C51F-39A6-6052-0A7E5AD17161'}
				startPosition : PositionXYC;
	END_VAR
END_METHOD


	(* Get the end position of the segment. *)
	METHOD GetEndPosition
	VAR_IN_OUT
		(* The current end position of the segment. *)
 {attribute 'GUID' := 'CB2F0EE9-C51F-39A6-6052-0A7E5AD17161'}
				endPosition : PositionXYC;
	END_VAR
END_METHOD


	(* Get a position on the path at a specific arclength value. *)
	METHOD GetPositionAt
	VAR_INPUT
		(* Arc length value where the position is evaluated. *)
		arcLength : LREAL;
	END_VAR
	VAR_IN_OUT
		(* The position at the specified arc parameter. *)
 {attribute 'GUID' := 'CB2F0EE9-C51F-39A6-6052-0A7E5AD17161'}
				position : PositionXYC;
	END_VAR
END_METHOD


	(* Get the dynamic information when moving along a path
				    with specific arclength value and dynamic changes. *)
	METHOD GetStateAt
	VAR_INPUT
		(* Arc length value where the position is evaluated. *)
		arcLength : LREAL;
		(* Velocity of the arc length parameter. *)
		arcVelocity : LREAL;
		(* Acceleration of the arc length parameter. *)
		arcAcceleration : LREAL;
	END_VAR
	VAR_IN_OUT
		(* The position at the specified arc parameter. *)
 {attribute 'GUID' := 'CB2F0EE9-C51F-39A6-6052-0A7E5AD17161'}
				position : PositionXYC;
		(* The velocity at the specified dynamic state. *)
 {attribute 'GUID' := '7FF54AC7-5E94-3451-6B65-C705B395D66F'}
				velocity : TangentXYC;
		(* The acceleration at the specified dynamic state. *)
 {attribute 'GUID' := '7FF54AC7-5E94-3451-6B65-C705B395D66F'}
				acceleration : TangentXYC;
	END_VAR
END_METHOD

END_FUNCTION_BLOCK

// POUs/Shapes/Geometry3D/Container3D

	{attribute 'c++_compatible'}
	{attribute 'external_name' := 'Container3D_GUID_48B68479_3BDD_3C93_5DE0_962FAE1B301D'}
	{attribute 'TcIecLibraryType'}
	{attribute 'no_explicit_call' :='do not call this POU directly'}
	{attribute 'no_assign'}
	FUNCTION_BLOCK Container3D EXTENDS Geometry3D


	(* Internal method *)
	METHOD FB_init : BOOL
	VAR_INPUT
		(*  if TRUE, the retain variables are initialized (warm start / cold start) *)
		bInitRetains : BOOL;
		(*  if TRUE, the instance afterwards gets moved into the copy code (online change) *)
		bInCopyCode : BOOL;
	END_VAR
END_METHOD


	(* Internal method *)
	{attribute 'hide'}
	METHOD FB_exit : BOOL
	VAR_INPUT
		(*  if TRUE, the exit method is called for exiting an instance that is copied afterwards (online change). *)
		bInCopyCode : BOOL;
	END_VAR
END_METHOD


	(* Add a geometry to the container. *)
	METHOD AddElement : UDINT
	VAR_IN_OUT
		(* The geometry to add. *)
 {attribute 'GUID' := 'C95BAD6C-3403-3B7E-68DC-43483A58037D'}
				geometry : Geometry3D;
	END_VAR
END_METHOD


	(* Remove a specified geometry from the container. *)
	METHOD RemoveElement
	VAR_INPUT
		(* Identifier of the geometry to remove. *)
		id : UDINT;
	END_VAR
END_METHOD


	(* Remove all geometries from container. *)
	METHOD Clear
END_METHOD


	(* Get the number of geometry elements in container. *)
	METHOD GetCount : UDINT
END_METHOD

END_FUNCTION_BLOCK

// POUs/Shapes/Geometry3D/Extrude3D

	{attribute 'c++_compatible'}
	{attribute 'external_name' := 'Extrude3D_GUID_024E4576_FB1B_3FDF_59B6_AFE80F47B286'}
	{attribute 'TcIecLibraryType'}
	{attribute 'no_explicit_call' :='do not call this POU directly'}
	{attribute 'no_assign'}
	FUNCTION_BLOCK Extrude3D EXTENDS Geometry3D


	(* Internal method *)
	METHOD FB_init : BOOL
	VAR_INPUT
		(*  if TRUE, the retain variables are initialized (warm start / cold start) *)
		bInitRetains : BOOL;
		(*  if TRUE, the instance afterwards gets moved into the copy code (online change) *)
		bInCopyCode : BOOL;
	END_VAR
END_METHOD


	(* Internal method *)
	{attribute 'hide'}
	METHOD FB_exit : BOOL
	VAR_INPUT
		(*  if TRUE, the exit method is called for exiting an instance that is copied afterwards (online change). *)
		bInCopyCode : BOOL;
	END_VAR
END_METHOD


	(* Define the extrude geometry with a path and a array of xy-points *)
	METHOD DefineByPath : BOOL
	VAR_IN_OUT
		(* Cross section values *)
 {attribute 'GUID' := '4E15B754-A8FD-31E0-757D-498AD44094D3'}
				PointerToCrossSection : POINTER TO PositionXY;
	END_VAR
	VAR_INPUT
		(* Number of cross section points *)
		NumberOfCrossSectionPoints : UDINT;
	END_VAR
	VAR_IN_OUT
		(* The path *)
 {attribute 'GUID' := 'FAA4A218-6E85-313D-57C6-24F488D84AF1'}
				Path : PathXYZ;
	END_VAR
	VAR_INPUT
		(* Number of path points *)
		NumberOfPathPoints : UDINT;
	END_VAR
END_METHOD

END_FUNCTION_BLOCK

// POUs/Paths/Components/PathXYZ

	{attribute 'c++_compatible'}
	{attribute 'external_name' := 'PathXYZ_GUID_FAA4A218_6E85_313D_57C6_24F488D84AF1'}
	{attribute 'TcIecLibraryType'}
	{attribute 'no_explicit_call' :='do not call this POU directly'}
	{attribute 'no_assign'}
	(* A path in the xy-plane with an additional orientation at every path position. *)
	FUNCTION_BLOCK PathXYZ EXTENDS IPlcPath3D


	(* Internal method *)
	{attribute 'hide'}
	METHOD FB_init : BOOL
	VAR_INPUT
		(*  if TRUE, the retain variables are initialized (warm start / cold start) *)
		bInitRetains : BOOL;
		(*  if TRUE, the instance afterwards gets moved into the copy code (online change) *)
		bInCopyCode : BOOL;
	END_VAR
END_METHOD


	(* Internal method *)
	{attribute 'hide'}
	METHOD FB_exit : BOOL
	VAR_INPUT
		(*  if TRUE, the exit method is called for exiting an instance that is copied afterwards (online change). *)
		bInCopyCode : BOOL;
	END_VAR
END_METHOD


	(* Append a smooth transition from the current end of the path
				    to the specified position. *)
	METHOD AppendPosition
	VAR_IN_OUT
		(* The position to append. *)
 {attribute 'GUID' := 'F25F0046-C763-3F00-5FBE-159880852C99'}
				position : Position3D;
	END_VAR
END_METHOD


	(* Append a smooth transition from the current end of the path
				    to the specified position. *)
	METHOD AppendPositionXYZ
	VAR_INPUT
		(* x-component of the position to append. *)
		x : LREAL;
		(* y-component of the position to append. *)
		y : LREAL;
		(* z-component of the position to append. *)
		c : LREAL;
	END_VAR
END_METHOD


	(* Append a line to this path. *)
	METHOD AppendLine
	VAR_IN_OUT
		(* Start position of the line. *)
 {attribute 'GUID' := 'F25F0046-C763-3F00-5FBE-159880852C99'}
				startPos : Position3D;
		(* End position of the line. *)
 {attribute 'GUID' := 'F25F0046-C763-3F00-5FBE-159880852C99'}
				endPos : Position3D;
	END_VAR
END_METHOD


	(* Append a smooth transition from the current end of the path
				    to the specified position. *)
	METHOD AppendLineXYZ
	VAR_INPUT
		(* x-component of the start position. *)
		x0 : LREAL;
		(* y-component of the start position. *)
		y0 : LREAL;
		(* z-component of the start position. *)
		z0 : LREAL;
		(* x-component of the end position. *)
		x1 : LREAL;
		(* y-component of the end position. *)
		y1 : LREAL;
		(* z-component of the end position. *)
		z1 : LREAL;
	END_VAR
END_METHOD


	(* Append a circle to this path. *)
	METHOD AppendCircle
	VAR_IN_OUT
		(* Start position of the circle. *)
 {attribute 'GUID' := 'F25F0046-C763-3F00-5FBE-159880852C99'}
				startPos : Position3D;
		(* End position of the circle. *)
 {attribute 'GUID' := 'F25F0046-C763-3F00-5FBE-159880852C99'}
				endPos : Position3D;
		(* Center of the circle. *)
 {attribute 'GUID' := '4E15B754-A8FD-31E0-757D-498AD44094D3'}
				center : PositionXY;
	END_VAR
	VAR_INPUT
		(* Set whether the circle runs clockwise or counter-clockwise. *)
		clockwise : BOOL;
	END_VAR
END_METHOD


	(* Append a smooth transition from the current end of the path
				    to the specified position with tangent. *)
	METHOD AppendPositionTangent
	VAR_IN_OUT
		(* The position to append. *)
 {attribute 'GUID' := 'F25F0046-C763-3F00-5FBE-159880852C99'}
				position : Position3D;
		(* The tangent to append *)
 {attribute 'GUID' := '2D21607C-3841-350E-4823-AED297AC450B'}
				tangent : Tangent3D;
	END_VAR
END_METHOD


	(* Get the start position of the path. *)
	METHOD GetStartPosition
	VAR_IN_OUT
		(* The current start position of the path. *)
 {attribute 'GUID' := 'F25F0046-C763-3F00-5FBE-159880852C99'}
				startPosition : Position3D;
	END_VAR
END_METHOD


	(* Get the end position of the segment. *)
	METHOD GetEndPosition
	VAR_IN_OUT
		(* The current end position of the segment. *)
 {attribute 'GUID' := 'F25F0046-C763-3F00-5FBE-159880852C99'}
				endPosition : Position3D;
	END_VAR
END_METHOD


	(* Get a position on the path at a specific arclength value. *)
	METHOD GetPositionAt
	VAR_INPUT
		(* Arc length value where the position is evaluated. *)
		arcLength : LREAL;
	END_VAR
	VAR_IN_OUT
		(* The position at the specified arc parameter. *)
 {attribute 'GUID' := 'F25F0046-C763-3F00-5FBE-159880852C99'}
				position : Position3D;
	END_VAR
END_METHOD


	(* Get the dynamic information when moving along a path
				    with specific arclength value and dynamic changes. *)
	METHOD GetStateAt
	VAR_INPUT
		(* Arc length value where the position is evaluated. *)
		arcLength : LREAL;
		(* Velocity of the arc length parameter. *)
		arcVelocity : LREAL;
		(* Acceleration of the arc length parameter. *)
		arcAcceleration : LREAL;
	END_VAR
	VAR_IN_OUT
		(* The position at the specified arc parameter. *)
 {attribute 'GUID' := 'F25F0046-C763-3F00-5FBE-159880852C99'}
				position : Position3D;
		(* The velocity at the specified dynamic state. *)
 {attribute 'GUID' := '2D21607C-3841-350E-4823-AED297AC450B'}
				velocity : Tangent3D;
		(* The acceleration at the specified dynamic state. *)
 {attribute 'GUID' := '2D21607C-3841-350E-4823-AED297AC450B'}
				acceleration : Tangent3D;
	END_VAR
END_METHOD

END_FUNCTION_BLOCK

// POUs/Paths/Components/PathXY

	{attribute 'c++_compatible'}
	{attribute 'external_name' := 'PathXY_GUID_1D433863_0502_3FD3_78D8_960BB49E6AC8'}
	{attribute 'TcIecLibraryType'}
	{attribute 'no_explicit_call' :='do not call this POU directly'}
	{attribute 'no_assign'}
	(* A path in the xy-plane. *)
	FUNCTION_BLOCK PathXY EXTENDS IPlcPath2D


	(* Internal method *)
	{attribute 'hide'}
	METHOD FB_init : BOOL
	VAR_INPUT
		(*  if TRUE, the retain variables are initialized (warm start / cold start) *)
		bInitRetains : BOOL;
		(*  if TRUE, the instance afterwards gets moved into the copy code (online change) *)
		bInCopyCode : BOOL;
	END_VAR
END_METHOD


	(* Internal method *)
	{attribute 'hide'}
	METHOD FB_exit : BOOL
	VAR_INPUT
		(*  if TRUE, the exit method is called for exiting an instance that is copied afterwards (online change). *)
		bInCopyCode : BOOL;
	END_VAR
END_METHOD


	(* Append a smooth transition from the current end of the path
				    to the specified position. *)
	METHOD AppendPosition
	VAR_IN_OUT
		(* The position to append. *)
 {attribute 'GUID' := '4E15B754-A8FD-31E0-757D-498AD44094D3'}
				position : PositionXY;
	END_VAR
END_METHOD


	(* Append a smooth transition from the current end of the path
				    to the specified position. *)
	METHOD AppendPositionXY
	VAR_INPUT
		(* x-component of the position to append. *)
		x : LREAL;
		(* y-component of the position to append. *)
		y : LREAL;
	END_VAR
END_METHOD


	(* Append a line to this path. *)
	METHOD AppendLine
	VAR_IN_OUT
		(* Start position of the line. *)
 {attribute 'GUID' := '4E15B754-A8FD-31E0-757D-498AD44094D3'}
				startPos : PositionXY;
		(* End position of the line. *)
 {attribute 'GUID' := '4E15B754-A8FD-31E0-757D-498AD44094D3'}
				endPos : PositionXY;
	END_VAR
END_METHOD


	(* Append a circle to this path. *)
	METHOD AppendCircle
	VAR_IN_OUT
		(* Start position of the circle. *)
 {attribute 'GUID' := '4E15B754-A8FD-31E0-757D-498AD44094D3'}
				startPos : PositionXY;
		(* End position of the circle. *)
 {attribute 'GUID' := '4E15B754-A8FD-31E0-757D-498AD44094D3'}
				endPos : PositionXY;
		(* Center of the circle. *)
 {attribute 'GUID' := '4E15B754-A8FD-31E0-757D-498AD44094D3'}
				center : PositionXY;
	END_VAR
	VAR_INPUT
		(* Set whether the circle runs clockwise or counter-clockwise. *)
		clockwise : BOOL;
	END_VAR
END_METHOD


	(* Get the start position of the path. *)
	METHOD GetStartPosition
	VAR_IN_OUT
		(* The current start position of the path. *)
 {attribute 'GUID' := '4E15B754-A8FD-31E0-757D-498AD44094D3'}
				startPosition : PositionXY;
	END_VAR
END_METHOD


	(* Get the end position of the segment. *)
	METHOD GetEndPosition
	VAR_IN_OUT
		(* The current end position of the segment. *)
 {attribute 'GUID' := '4E15B754-A8FD-31E0-757D-498AD44094D3'}
				endPosition : PositionXY;
	END_VAR
END_METHOD


	(* Get a position on the path at a specific arclength value. *)
	METHOD GetPositionAt
	VAR_INPUT
		(* Arc length value where the position is evaluated. *)
		arcLength : LREAL;
	END_VAR
	VAR_IN_OUT
		(* The position at the specified arc parameter. *)
 {attribute 'GUID' := '4E15B754-A8FD-31E0-757D-498AD44094D3'}
				position : PositionXY;
	END_VAR
END_METHOD


	(* Get the dynamic information when moving along a path
				    with specific arclength value and dynamic changes. *)
	METHOD GetStateAt
	VAR_INPUT
		(* Arc length value where the position is evaluated. *)
		arcLength : LREAL;
		(* Velocity of the arc length parameter. *)
		arcVelocity : LREAL;
		(* Acceleration of the arc length parameter. *)
		arcAcceleration : LREAL;
	END_VAR
	VAR_IN_OUT
		(* The position at the specified arc parameter. *)
 {attribute 'GUID' := '4E15B754-A8FD-31E0-757D-498AD44094D3'}
				position : PositionXY;
		(* The velocity at the specified dynamic state. *)
 {attribute 'GUID' := 'FE5FBEA1-CCA0-3BC6-7207-1BBF2A5405AC'}
				velocity : TangentXY;
		(* The acceleration at the specified dynamic state. *)
 {attribute 'GUID' := 'FE5FBEA1-CCA0-3BC6-7207-1BBF2A5405AC'}
				acceleration : TangentXY;
	END_VAR
END_METHOD

END_FUNCTION_BLOCK

// POUs/Shapes/Geometry2D/1D/Line2D

	{attribute 'c++_compatible'}
	{attribute 'external_name' := 'Line2D_GUID_09CA5A70_D489_376A_74DF_E7C2BC140EEA'}
	{attribute 'TcIecLibraryType'}
	{attribute 'no_explicit_call' :='do not call this POU directly'}
	{attribute 'no_assign'}
	(* 2D Geometry Line *)
	FUNCTION_BLOCK Line2D EXTENDS Geometry2D


	(* Internal method *)
	METHOD FB_init : BOOL
	VAR_INPUT
		(*  if TRUE, the retain variables are initialized (warm start / cold start) *)
		bInitRetains : BOOL;
		(*  if TRUE, the instance afterwards gets moved into the copy code (online change) *)
		bInCopyCode : BOOL;
	END_VAR
END_METHOD


	(* Internal method *)
	{attribute 'hide'}
	METHOD FB_exit : BOOL
	VAR_INPUT
		(*  if TRUE, the exit method is called for exiting an instance that is copied afterwards (online change). *)
		bInCopyCode : BOOL;
	END_VAR
END_METHOD


	(* Define a line by two positions. *)
	METHOD DefineByPositions
	VAR_IN_OUT
		(* 1st position on the line to define. *)
 {attribute 'GUID' := '4E15B754-A8FD-31E0-757D-498AD44094D3'}
				position0 : PositionXY;
		(* 2nd position on the line to define. *)
 {attribute 'GUID' := '4E15B754-A8FD-31E0-757D-498AD44094D3'}
				position1 : PositionXY;
	END_VAR
END_METHOD


	(* Define a line by a position on the line and its direction. *)
	METHOD DefineByDirection
	VAR_IN_OUT
		(* Position on the line *)
 {attribute 'GUID' := '4E15B754-A8FD-31E0-757D-498AD44094D3'}
				position : PositionXY;
		(* Direction of the line *)
 {attribute 'GUID' := 'FE5FBEA1-CCA0-3BC6-7207-1BBF2A5405AC'}
				direction : TangentXY;
	END_VAR
END_METHOD


	(* Set the direction of the line. *)
	METHOD SetDirection
	VAR_IN_OUT
		(* The direction to set. *)
 {attribute 'GUID' := 'FE5FBEA1-CCA0-3BC6-7207-1BBF2A5405AC'}
				direction : TangentXY;
	END_VAR
END_METHOD


	(* Get the direction of the line. *)
	METHOD GetDirection
	VAR_IN_OUT
		(* The current direction of the line. *)
 {attribute 'GUID' := 'FE5FBEA1-CCA0-3BC6-7207-1BBF2A5405AC'}
				direction : TangentXY;
	END_VAR
END_METHOD


	(* Get a position on the line at a specific arclength value. *)
	METHOD GetPositionAt
	VAR_INPUT
		(* Arc length value where the position is evaluated. *)
		arcLength : LREAL;
	END_VAR
	VAR_IN_OUT
		(* The position at the specified arc parameter. *)
 {attribute 'GUID' := 'CB2F0EE9-C51F-39A6-6052-0A7E5AD17161'}
				position : PositionXYC;
	END_VAR
END_METHOD

END_FUNCTION_BLOCK

// POUs/Shapes/Geometry2D/1D/Segment2D

	{attribute 'c++_compatible'}
	{attribute 'external_name' := 'Segment2D_GUID_683BBA75_D50F_3F74_7789_921214589D30'}
	{attribute 'TcIecLibraryType'}
	{attribute 'no_explicit_call' :='do not call this POU directly'}
	{attribute 'no_assign'}
	FUNCTION_BLOCK Segment2D EXTENDS Geometry2D


	(* Internal method *)
	METHOD FB_init : BOOL
	VAR_INPUT
		(*  if TRUE, the retain variables are initialized (warm start / cold start) *)
		bInitRetains : BOOL;
		(*  if TRUE, the instance afterwards gets moved into the copy code (online change) *)
		bInCopyCode : BOOL;
	END_VAR
END_METHOD


	(* Internal method *)
	{attribute 'hide'}
	METHOD FB_exit : BOOL
	VAR_INPUT
		(*  if TRUE, the exit method is called for exiting an instance that is copied afterwards (online change). *)
		bInCopyCode : BOOL;
	END_VAR
END_METHOD


	(* Set the start position of the segment. *)
	METHOD SetStartPosition
	VAR_IN_OUT
		(* Start position of the segment to set. *)
 {attribute 'GUID' := '4E15B754-A8FD-31E0-757D-498AD44094D3'}
				startPos : PositionXY;
	END_VAR
END_METHOD


	(* Set the start position of the segment. *)
	METHOD SetStartPositionXY
	VAR_INPUT
		(* x-component of the start position. *)
		x : LREAL;
		(* y-component of the start position. *)
		y : LREAL;
	END_VAR
END_METHOD


	(* Set the end position of the segment. *)
	METHOD SetEndPosition
	VAR_IN_OUT
		(* End position of the segment to set. *)
 {attribute 'GUID' := '4E15B754-A8FD-31E0-757D-498AD44094D3'}
				endPos : PositionXY;
	END_VAR
END_METHOD


	(* Set the end position of the segment. *)
	METHOD SetEndPositionXY
	VAR_INPUT
		(* x-component of the end position. *)
		x : LREAL;
		(* y-component of the end position. *)
		y : LREAL;
	END_VAR
END_METHOD


	(* Get the x-component of the segment length in respect to the root coordinate system. *)
	METHOD Get_dX : LREAL
END_METHOD


	(* Get the y-component of the segment length in respect to the root coordinate system. *)
	METHOD Get_dY : LREAL
END_METHOD


	(* Get the length of the segment. *)
	METHOD GetLength : LREAL
END_METHOD


	(* Get the start position of the segment. *)
	METHOD GetStartPosition
	VAR_IN_OUT
		(* The current start position of the segment. *)
 {attribute 'GUID' := '4E15B754-A8FD-31E0-757D-498AD44094D3'}
				startPosition : PositionXY;
	END_VAR
END_METHOD


	(* Get the end position of the segment. *)
	METHOD GetEndPosition
	VAR_IN_OUT
		(* The current end position of the segment. *)
 {attribute 'GUID' := '4E15B754-A8FD-31E0-757D-498AD44094D3'}
				endPosition : PositionXY;
	END_VAR
END_METHOD


	(* Get the direction of the segment. *)
	METHOD GetDirection
	VAR_IN_OUT
		(* The current direction of the segment. *)
 {attribute 'GUID' := 'FE5FBEA1-CCA0-3BC6-7207-1BBF2A5405AC'}
				direction : TangentXY;
	END_VAR
END_METHOD


	(* Get a position on the segment at a specific arclength value. *)
	METHOD GetPositionAt
	VAR_INPUT
		(* Arc length value where the position is evaluated. *)
		arcLength : LREAL;
	END_VAR
	VAR_IN_OUT
		(* The position at the specified arc parameter. *)
 {attribute 'GUID' := 'CB2F0EE9-C51F-39A6-6052-0A7E5AD17161'}
				position : PositionXYC;
	END_VAR
END_METHOD

END_FUNCTION_BLOCK

// POUs/Shapes/Geometry2D/1D/Circle2D

	{attribute 'c++_compatible'}
	{attribute 'external_name' := 'Circle2D_GUID_3F7C6906_D993_3CBD_4553_B02232F1D891'}
	{attribute 'TcIecLibraryType'}
	{attribute 'no_explicit_call' :='do not call this POU directly'}
	{attribute 'no_assign'}
	FUNCTION_BLOCK Circle2D EXTENDS Geometry2D


	(* Internal method *)
	METHOD FB_init : BOOL
	VAR_INPUT
		(*  if TRUE, the retain variables are initialized (warm start / cold start) *)
		bInitRetains : BOOL;
		(*  if TRUE, the instance afterwards gets moved into the copy code (online change) *)
		bInCopyCode : BOOL;
	END_VAR
END_METHOD


	(* Internal method *)
	{attribute 'hide'}
	METHOD FB_exit : BOOL
	VAR_INPUT
		(*  if TRUE, the exit method is called for exiting an instance that is copied afterwards (online change). *)
		bInCopyCode : BOOL;
	END_VAR
END_METHOD


	(* Get the length of the circle. *)
	METHOD GetLength : LREAL
END_METHOD


	(* Get a position on the circle at a specific arclength value. *)
	METHOD GetPositionAt
	VAR_INPUT
		(* Arc length value where the position is evaluated. *)
		arcLength : LREAL;
	END_VAR
	VAR_IN_OUT
		(* The position at the specified arc parameter. *)
 {attribute 'GUID' := 'CB2F0EE9-C51F-39A6-6052-0A7E5AD17161'}
				position : PositionXYC;
	END_VAR
END_METHOD


	PROPERTY radius : LREAL
GET
END_GET
SET
END_SET
END_PROPERTY

END_FUNCTION_BLOCK

// POUs/Shapes/Geometry2D/2D/Disc2D

	{attribute 'c++_compatible'}
	{attribute 'external_name' := 'Disc2D_GUID_C28B15E8_4748_354B_5D11_3B4336E0DDBD'}
	{attribute 'TcIecLibraryType'}
	{attribute 'no_explicit_call' :='do not call this POU directly'}
	{attribute 'no_assign'}
	FUNCTION_BLOCK Disc2D EXTENDS Geometry2D


	(* Internal method *)
	METHOD FB_init : BOOL
	VAR_INPUT
		(*  if TRUE, the retain variables are initialized (warm start / cold start) *)
		bInitRetains : BOOL;
		(*  if TRUE, the instance afterwards gets moved into the copy code (online change) *)
		bInCopyCode : BOOL;
	END_VAR
END_METHOD


	(* Internal method *)
	{attribute 'hide'}
	METHOD FB_exit : BOOL
	VAR_INPUT
		(*  if TRUE, the exit method is called for exiting an instance that is copied afterwards (online change). *)
		bInCopyCode : BOOL;
	END_VAR
END_METHOD


	(* Get the area of the disc. *)
	METHOD GetArea : LREAL
END_METHOD


	PROPERTY radius : LREAL
GET
END_GET
SET
END_SET
END_PROPERTY

END_FUNCTION_BLOCK

// POUs/Shapes/Geometry2D/2D/Rectangle2D

	{attribute 'c++_compatible'}
	{attribute 'external_name' := 'Rectangle2D_GUID_ECA92675_C32D_3903_46C9_804A2B07F2AF'}
	{attribute 'TcIecLibraryType'}
	{attribute 'no_explicit_call' :='do not call this POU directly'}
	{attribute 'no_assign'}
	FUNCTION_BLOCK Rectangle2D EXTENDS Geometry2D


	(* Internal method *)
	METHOD FB_init : BOOL
	VAR_INPUT
		(*  if TRUE, the retain variables are initialized (warm start / cold start) *)
		bInitRetains : BOOL;
		(*  if TRUE, the instance afterwards gets moved into the copy code (online change) *)
		bInCopyCode : BOOL;
	END_VAR
END_METHOD


	(* Internal method *)
	{attribute 'hide'}
	METHOD FB_exit : BOOL
	VAR_INPUT
		(*  if TRUE, the exit method is called for exiting an instance that is copied afterwards (online change). *)
		bInCopyCode : BOOL;
	END_VAR
END_METHOD


	(* Set the dimensions of the rectangle. *)
	METHOD SetDimensions
	VAR_INPUT
		(* The width of the rectangle to set. *)
		width : LREAL;
		(* The height of the rectangle to set. *)
		height : LREAL;
	END_VAR
END_METHOD


	(* Get the area of the rectangle. *)
	METHOD GetArea : LREAL
END_METHOD


	PROPERTY width : LREAL
GET
END_GET
SET
END_SET
END_PROPERTY


	PROPERTY height : LREAL
GET
END_GET
SET
END_SET
END_PROPERTY

END_FUNCTION_BLOCK

// POUs/Shapes/Geometry2D/Functions/CheckCollision2D

	{attribute 'TcIecLibraryType'}
	{attribute 'external_name' := 'CheckCollision2D_GUID_521AB9F2_59D4_32FD_4B8B_1872AF58C22B'}
	(* Check if two geometries are currently colliding. *)
	FUNCTION CheckCollision2D : BOOL
	VAR_IN_OUT
		geometry0	:	IPlcGeometry2D;	(* 1st input geometry to check for collision. *)
		geometry1	:	IPlcGeometry2D;	(* 2nd input geometry to check of collision. *)
	END_VAR

END_FUNCTION

// POUs/Shapes/Geometry2D/Functions/GetDistance2D

	{attribute 'TcIecLibraryType'}
	{attribute 'external_name' := 'GetDistance2D_GUID_6DD5C20A_98AF_3868_7FC7_16531AE31FB7'}
	(* Get the distance between two geometries. *)
	FUNCTION GetDistance2D : LREAL
	VAR_IN_OUT
		geometry0	:	IPlcGeometry2D;	(* 1st input geometry to calculate the distance of. *)
		geometry1	:	IPlcGeometry2D;	(* 2nd input geometry to calculate the distance of. *)
	END_VAR

END_FUNCTION

// POUs/Shapes/Geometry2D/Functions/GetLinkingLine2D

	{attribute 'TcIecLibraryType'}
	{attribute 'external_name' := 'GetLinkingLine2D_GUID_2B3EC235_EA59_3605_5BB9_79C853CFB0E1'}
	(* Get the shortest path between two geometries. *)
	FUNCTION GetLinkingLine2D : BOOL
	VAR_IN_OUT
		geometry0	:	IPlcGeometry2D;	(* 1st input geometry to calculate the linking line for. *)
		geometry1	:	IPlcGeometry2D;	(* 2nd input geometry to calculate the linking line for. *)
		linkingLine	:	Segment2D;	(* Return the resulting linking line. *)
	END_VAR

END_FUNCTION

// POUs/Shapes/Geometry3D/1D/Line3D

	{attribute 'c++_compatible'}
	{attribute 'external_name' := 'Line3D_GUID_047421FF_867C_3F96_5D46_8242E88216F1'}
	{attribute 'TcIecLibraryType'}
	{attribute 'no_explicit_call' :='do not call this POU directly'}
	{attribute 'no_assign'}
	(* 3D Geometry Line *)
	FUNCTION_BLOCK Line3D EXTENDS Geometry3D


	(* Internal method *)
	METHOD FB_init : BOOL
	VAR_INPUT
		(*  if TRUE, the retain variables are initialized (warm start / cold start) *)
		bInitRetains : BOOL;
		(*  if TRUE, the instance afterwards gets moved into the copy code (online change) *)
		bInCopyCode : BOOL;
	END_VAR
END_METHOD


	(* Internal method *)
	{attribute 'hide'}
	METHOD FB_exit : BOOL
	VAR_INPUT
		(*  if TRUE, the exit method is called for exiting an instance that is copied afterwards (online change). *)
		bInCopyCode : BOOL;
	END_VAR
END_METHOD


	(* Define a line by two positions. *)
	METHOD DefineByPositions
	VAR_IN_OUT
		(* 1st position on the line to define. *)
 {attribute 'GUID' := 'F25F0046-C763-3F00-5FBE-159880852C99'}
				position0 : Position3D;
		(* 2nd position on the line to define. *)
 {attribute 'GUID' := 'F25F0046-C763-3F00-5FBE-159880852C99'}
				position1 : Position3D;
	END_VAR
END_METHOD


	(* Define a line by a position on the line and its direction. *)
	METHOD DefineByDirection
	VAR_IN_OUT
		(* Position on the line. *)
 {attribute 'GUID' := 'F25F0046-C763-3F00-5FBE-159880852C99'}
				position : Position3D;
		(* Direction of the line. *)
 {attribute 'GUID' := '2D21607C-3841-350E-4823-AED297AC450B'}
				direction : Tangent3D;
	END_VAR
END_METHOD


	(* Set the direction of the line. *)
	METHOD SetDirection
	VAR_IN_OUT
		(* The direction to set. *)
 {attribute 'GUID' := '2D21607C-3841-350E-4823-AED297AC450B'}
				direction : Tangent3D;
	END_VAR
END_METHOD


	(* Get the direction of the line. *)
	METHOD GetDirection
	VAR_IN_OUT
		(* The current direction of the line. *)
 {attribute 'GUID' := '2D21607C-3841-350E-4823-AED297AC450B'}
				direction : Tangent3D;
	END_VAR
END_METHOD


	(* Get a position on the line at a specific arclength value. *)
	METHOD GetPositionAt
	VAR_INPUT
		(* Arc length value where the position is evaluated. *)
		arcLength : LREAL;
	END_VAR
	VAR_IN_OUT
		(* The position at the specified arc parameter. *)
 {attribute 'GUID' := 'D2337217-563D-354C-4349-0B99B7C3F40C'}
				position : PositionSE3;
	END_VAR
END_METHOD

END_FUNCTION_BLOCK

// POUs/Shapes/Geometry3D/1D/Segment3D

	{attribute 'c++_compatible'}
	{attribute 'external_name' := 'Segment3D_GUID_39A5336D_3980_38B2_456F_FDF60F12D6A1'}
	{attribute 'TcIecLibraryType'}
	{attribute 'no_explicit_call' :='do not call this POU directly'}
	{attribute 'no_assign'}
	FUNCTION_BLOCK Segment3D EXTENDS Geometry3D


	(* Internal method *)
	METHOD FB_init : BOOL
	VAR_INPUT
		(*  if TRUE, the retain variables are initialized (warm start / cold start) *)
		bInitRetains : BOOL;
		(*  if TRUE, the instance afterwards gets moved into the copy code (online change) *)
		bInCopyCode : BOOL;
	END_VAR
END_METHOD


	(* Internal method *)
	{attribute 'hide'}
	METHOD FB_exit : BOOL
	VAR_INPUT
		(*  if TRUE, the exit method is called for exiting an instance that is copied afterwards (online change). *)
		bInCopyCode : BOOL;
	END_VAR
END_METHOD


	(* Set the start position of the segment. *)
	METHOD SetStartPosition
	VAR_IN_OUT
		(* Start position of the segment to set. *)
 {attribute 'GUID' := 'F25F0046-C763-3F00-5FBE-159880852C99'}
				startPos : Position3D;
	END_VAR
END_METHOD


	(* Set the start position of the segment. *)
	METHOD SetStartPositionXYZ
	VAR_INPUT
		(* x-component of the start position. *)
		x : LREAL;
		(* y-component of the start position. *)
		y : LREAL;
		(* z-component of the start position. *)
		z : LREAL;
	END_VAR
END_METHOD


	(* Set the end position of the segment. *)
	METHOD SetEndPosition
	VAR_IN_OUT
		(* End position of the segment to set. *)
 {attribute 'GUID' := 'F25F0046-C763-3F00-5FBE-159880852C99'}
				endPos : Position3D;
	END_VAR
END_METHOD


	(* Set the end position of the segment. *)
	METHOD SetEndPositionXYZ
	VAR_INPUT
		(* x-component of the end position. *)
		x : LREAL;
		(* y-component of the end position. *)
		y : LREAL;
		(* z-component of the end position. *)
		z : LREAL;
	END_VAR
END_METHOD


	(* Get the x-component of the segment length in respect to the root coordinate system. *)
	METHOD Get_dX : LREAL
END_METHOD


	(* Get the y-component of the segment length in respect to the root coordinate system. *)
	METHOD Get_dY : LREAL
END_METHOD


	(* Get the z-component of the segment length in respect to the root coordinate system. *)
	METHOD Get_dZ : LREAL
END_METHOD


	(* Get the length of the segment. *)
	METHOD GetLength : LREAL
END_METHOD


	(* Get the start position of the segment. *)
	METHOD GetStartPosition
	VAR_IN_OUT
		(* The current start position of the segment. *)
 {attribute 'GUID' := 'F25F0046-C763-3F00-5FBE-159880852C99'}
				startPosition : Position3D;
	END_VAR
END_METHOD


	(* Get the end position of the segment. *)
	METHOD GetEndPosition
	VAR_IN_OUT
		(* The current end position of the segment. *)
 {attribute 'GUID' := 'F25F0046-C763-3F00-5FBE-159880852C99'}
				endPosition : Position3D;
	END_VAR
END_METHOD


	(* Get the direction of the segment. *)
	METHOD GetDirection
	VAR_IN_OUT
		(* The current direction of the segment. *)
 {attribute 'GUID' := '2D21607C-3841-350E-4823-AED297AC450B'}
				direction : Tangent3D;
	END_VAR
END_METHOD


	(* Get a position on the segment at a specific arclength value. *)
	METHOD GetPositionAt
	VAR_INPUT
		(* Arc length value where the position is evaluated. *)
		arcLength : LREAL;
	END_VAR
	VAR_IN_OUT
		(* The position at the specified arc parameter. *)
 {attribute 'GUID' := 'D2337217-563D-354C-4349-0B99B7C3F40C'}
				position : PositionSE3;
	END_VAR
END_METHOD

END_FUNCTION_BLOCK

// POUs/Shapes/Geometry3D/1D/Circle3D

	{attribute 'c++_compatible'}
	{attribute 'external_name' := 'Circle3D_GUID_F113EB8A_056E_380C_51D6_6FCC3A1B62CC'}
	{attribute 'TcIecLibraryType'}
	{attribute 'no_explicit_call' :='do not call this POU directly'}
	{attribute 'no_assign'}
	FUNCTION_BLOCK Circle3D EXTENDS Geometry3D


	(* Internal method *)
	METHOD FB_init : BOOL
	VAR_INPUT
		(*  if TRUE, the retain variables are initialized (warm start / cold start) *)
		bInitRetains : BOOL;
		(*  if TRUE, the instance afterwards gets moved into the copy code (online change) *)
		bInCopyCode : BOOL;
	END_VAR
END_METHOD


	(* Internal method *)
	{attribute 'hide'}
	METHOD FB_exit : BOOL
	VAR_INPUT
		(*  if TRUE, the exit method is called for exiting an instance that is copied afterwards (online change). *)
		bInCopyCode : BOOL;
	END_VAR
END_METHOD


	(* Set the normal vector of the circle. *)
	METHOD SetNormal
	VAR_IN_OUT
		(* Normal vector to set. *)
 {attribute 'GUID' := '2D21607C-3841-350E-4823-AED297AC450B'}
				normal : Tangent3D;
	END_VAR
END_METHOD


	(* Get the length of the circle. *)
	METHOD GetLength : LREAL
END_METHOD


	(* Get the normal vector of the circle. *)
	METHOD GetNormal
	VAR
		(* The current normal vector of the circle. *)
 {attribute 'GUID' := '2D21607C-3841-350E-4823-AED297AC450B'}
				normal : Tangent3D;
	END_VAR
END_METHOD


	(* Get a position on the circle at a specific arclength value. *)
	METHOD GetPositionAt
	VAR_INPUT
		(* Arc length value where the position is evaluated. *)
		arcLength : LREAL;
	END_VAR
	VAR_IN_OUT
		(* The position at the specified arc parameter. *)
 {attribute 'GUID' := 'D2337217-563D-354C-4349-0B99B7C3F40C'}
				position : PositionSE3;
	END_VAR
END_METHOD


	PROPERTY radius : LREAL
GET
END_GET
SET
END_SET
END_PROPERTY

END_FUNCTION_BLOCK

// POUs/Shapes/Geometry3D/2D/Plane3D

	{attribute 'c++_compatible'}
	{attribute 'external_name' := 'Plane3D_GUID_002309FB_0CE3_33DD_7AC8_37BC17A437D9'}
	{attribute 'TcIecLibraryType'}
	{attribute 'no_explicit_call' :='do not call this POU directly'}
	{attribute 'no_assign'}
	FUNCTION_BLOCK Plane3D EXTENDS Geometry3D


	(* Internal method *)
	METHOD FB_init : BOOL
	VAR_INPUT
		(*  if TRUE, the retain variables are initialized (warm start / cold start) *)
		bInitRetains : BOOL;
		(*  if TRUE, the instance afterwards gets moved into the copy code (online change) *)
		bInCopyCode : BOOL;
	END_VAR
END_METHOD


	(* Internal method *)
	{attribute 'hide'}
	METHOD FB_exit : BOOL
	VAR_INPUT
		(*  if TRUE, the exit method is called for exiting an instance that is copied afterwards (online change). *)
		bInCopyCode : BOOL;
	END_VAR
END_METHOD


	(* Set the normal of the plane. *)
	METHOD SetNormal
	VAR_IN_OUT
		(* The normal vector to set. *)
 {attribute 'GUID' := '2D21607C-3841-350E-4823-AED297AC450B'}
				normal : Tangent3D;
	END_VAR
END_METHOD


	(* Get the normal vector of the plane. *)
	METHOD GetNormal
	VAR
		(* The current normal vector of the plane. *)
 {attribute 'GUID' := '2D21607C-3841-350E-4823-AED297AC450B'}
				normal : Tangent3D;
	END_VAR
END_METHOD

END_FUNCTION_BLOCK

// POUs/Shapes/Geometry3D/2D/Disc3D

	{attribute 'c++_compatible'}
	{attribute 'external_name' := 'Disc3D_GUID_9A9DE724_9E00_3FC9_7066_600E76A2599B'}
	{attribute 'TcIecLibraryType'}
	{attribute 'no_explicit_call' :='do not call this POU directly'}
	{attribute 'no_assign'}
	FUNCTION_BLOCK Disc3D EXTENDS Geometry3D


	(* Internal method *)
	METHOD FB_init : BOOL
	VAR_INPUT
		(*  if TRUE, the retain variables are initialized (warm start / cold start) *)
		bInitRetains : BOOL;
		(*  if TRUE, the instance afterwards gets moved into the copy code (online change) *)
		bInCopyCode : BOOL;
	END_VAR
END_METHOD


	(* Internal method *)
	{attribute 'hide'}
	METHOD FB_exit : BOOL
	VAR_INPUT
		(*  if TRUE, the exit method is called for exiting an instance that is copied afterwards (online change). *)
		bInCopyCode : BOOL;
	END_VAR
END_METHOD


	(* Set the normal vector of the disc. *)
	METHOD SetNormal
	VAR_IN_OUT
		(* The normal to set. *)
 {attribute 'GUID' := '2D21607C-3841-350E-4823-AED297AC450B'}
				normal : Tangent3D;
	END_VAR
END_METHOD


	(* Get the normal vector of the disc. *)
	METHOD GetNormal
	VAR
		(* The current normal vector of the disc. *)
 {attribute 'GUID' := '2D21607C-3841-350E-4823-AED297AC450B'}
				normal : Tangent3D;
	END_VAR
END_METHOD


	(* Get the area of the disc. *)
	METHOD GetArea : LREAL
END_METHOD


	PROPERTY radius : LREAL
GET
END_GET
SET
END_SET
END_PROPERTY

END_FUNCTION_BLOCK

// POUs/Shapes/Geometry3D/2D/Rectangle3D

	{attribute 'c++_compatible'}
	{attribute 'external_name' := 'Rectangle3D_GUID_C8137469_4C86_375E_5260_CFBABC25F9A5'}
	{attribute 'TcIecLibraryType'}
	{attribute 'no_explicit_call' :='do not call this POU directly'}
	{attribute 'no_assign'}
	FUNCTION_BLOCK Rectangle3D EXTENDS Geometry3D


	(* Internal method *)
	METHOD FB_init : BOOL
	VAR_INPUT
		(*  if TRUE, the retain variables are initialized (warm start / cold start) *)
		bInitRetains : BOOL;
		(*  if TRUE, the instance afterwards gets moved into the copy code (online change) *)
		bInCopyCode : BOOL;
	END_VAR
END_METHOD


	(* Internal method *)
	{attribute 'hide'}
	METHOD FB_exit : BOOL
	VAR_INPUT
		(*  if TRUE, the exit method is called for exiting an instance that is copied afterwards (online change). *)
		bInCopyCode : BOOL;
	END_VAR
END_METHOD


	(* Set the dimensions of the rectangle. *)
	METHOD SetDimensions
	VAR_INPUT
		(* The width of the rectangle to set. *)
		width : LREAL;
		(* The height of the rectangle to set. *)
		height : LREAL;
	END_VAR
END_METHOD


	(* Get the area of the rectangle. *)
	METHOD GetArea : LREAL
END_METHOD


	PROPERTY width : LREAL
GET
END_GET
SET
END_SET
END_PROPERTY


	PROPERTY height : LREAL
GET
END_GET
SET
END_SET
END_PROPERTY

END_FUNCTION_BLOCK

// POUs/Shapes/Geometry3D/3D/Sphere3D

	{attribute 'c++_compatible'}
	{attribute 'external_name' := 'Sphere3D_GUID_32FB7944_121C_324F_4106_B133A80D99C7'}
	{attribute 'TcIecLibraryType'}
	{attribute 'no_explicit_call' :='do not call this POU directly'}
	{attribute 'no_assign'}
	FUNCTION_BLOCK Sphere3D EXTENDS Geometry3D


	(* Internal method *)
	METHOD FB_init : BOOL
	VAR_INPUT
		(*  if TRUE, the retain variables are initialized (warm start / cold start) *)
		bInitRetains : BOOL;
		(*  if TRUE, the instance afterwards gets moved into the copy code (online change) *)
		bInCopyCode : BOOL;
	END_VAR
END_METHOD


	(* Internal method *)
	{attribute 'hide'}
	METHOD FB_exit : BOOL
	VAR_INPUT
		(*  if TRUE, the exit method is called for exiting an instance that is copied afterwards (online change). *)
		bInCopyCode : BOOL;
	END_VAR
END_METHOD


	(* Get the volume of the sphere. *)
	METHOD GetVolume : LREAL
END_METHOD


	PROPERTY radius : LREAL
GET
END_GET
SET
END_SET
END_PROPERTY

END_FUNCTION_BLOCK

// POUs/Shapes/Geometry3D/3D/Cuboid3D

	{attribute 'c++_compatible'}
	{attribute 'external_name' := 'Cuboid3D_GUID_C0E1EDC7_67F3_3478_7B21_6FE899D11D6F'}
	{attribute 'TcIecLibraryType'}
	{attribute 'no_explicit_call' :='do not call this POU directly'}
	{attribute 'no_assign'}
	FUNCTION_BLOCK Cuboid3D EXTENDS Geometry3D


	(* Internal method *)
	METHOD FB_init : BOOL
	VAR_INPUT
		(* if TRUE, the retain variables are initialized (warm start / cold start) *)
		bInitRetains : BOOL;
		(* if TRUE, the instance afterwards gets moved into the copy code (online change) *)
		bInCopyCode : BOOL;
	END_VAR
END_METHOD


	(* Internal method *)
	{attribute 'hide'}
	METHOD FB_exit : BOOL
	VAR_INPUT
		(* if TRUE, the exit method is called for exiting an instance that is copied afterwards (online change). *)
		bInCopyCode : BOOL;
	END_VAR
END_METHOD


	(* Set the dimensions of the cuboid. *)
	METHOD SetDimensions
	VAR_INPUT
		(* local x-component *)
		length : LREAL;
		(* local y-component *)
		width : LREAL;
		(* local z-component *)
		height : LREAL;
	END_VAR
END_METHOD


	(* Get the volume of the cuboid. *)
	METHOD GetVolume : LREAL
END_METHOD


	PROPERTY length : LREAL
GET
END_GET
SET
END_SET
END_PROPERTY


	PROPERTY width : LREAL
GET
END_GET
SET
END_SET
END_PROPERTY


	PROPERTY height : LREAL
GET
END_GET
SET
END_SET
END_PROPERTY

END_FUNCTION_BLOCK

// POUs/Shapes/Geometry3D/3D/Cylinder3D

	{attribute 'c++_compatible'}
	{attribute 'external_name' := 'Cylinder3D_GUID_A47FB7FD_40DB_3C9A_6572_D123B8794DC8'}
	{attribute 'TcIecLibraryType'}
	{attribute 'no_explicit_call' :='do not call this POU directly'}
	{attribute 'no_assign'}
	FUNCTION_BLOCK Cylinder3D EXTENDS Geometry3D


	(* Internal method *)
	METHOD FB_init : BOOL
	VAR_INPUT
		(* if TRUE, the retain variables are initialized (warm start / cold start) *)
		bInitRetains : BOOL;
		(* if TRUE, the instance afterwards gets moved into the copy code (online change) *)
		bInCopyCode : BOOL;
	END_VAR
END_METHOD


	(* Internal method *)
	{attribute 'hide'}
	METHOD FB_exit : BOOL
	VAR_INPUT
		(* if TRUE, the exit method is called for exiting an instance that is copied afterwards (online change). *)
		bInCopyCode : BOOL;
	END_VAR
END_METHOD


	(* Set the dimensions of the cylinder. *)
	METHOD SetDimensions
	VAR_INPUT
		(* The radius to set. *)
		radius : LREAL;
		(* The height to set. *)
		height : LREAL;
	END_VAR
END_METHOD


	(* Get the volume of the cylinder. *)
	METHOD GetVolume : LREAL
END_METHOD


	PROPERTY radius : LREAL
GET
END_GET
SET
END_SET
END_PROPERTY


	PROPERTY height : LREAL
GET
END_GET
SET
END_SET
END_PROPERTY

END_FUNCTION_BLOCK

// POUs/Shapes/Geometry3D/Functions/CheckCollision3D

	{attribute 'TcIecLibraryType'}
	{attribute 'external_name' := 'CheckCollision3D_GUID_C79FB556_2CA7_3DA5_5EDD_D1693802375D'}
	(* Check if two geometries are currently colliding. *)
	FUNCTION CheckCollision3D : BOOL
	VAR_IN_OUT
		geometry0	:	IPlcGeometry3D;	(* 1st input geometry to check for collision. *)
		geometry1	:	IPlcGeometry3D;	(* 2nd input geometry to check of collision. *)
	END_VAR

END_FUNCTION

// POUs/Shapes/Geometry3D/Functions/GetDistance3D

	{attribute 'TcIecLibraryType'}
	{attribute 'external_name' := 'GetDistance3D_GUID_34268B43_BB7D_3AA1_71EA_013184AE62E5'}
	(* Get the distance between two geometries. *)
	FUNCTION GetDistance3D : LREAL
	VAR_IN_OUT
		geometry0	:	IPlcGeometry3D;	(* 1st input geometry to calculate the distance of. *)
		geometry1	:	IPlcGeometry3D;	(* 2nd input geometry to calculate the distance of. *)
	END_VAR

END_FUNCTION

// POUs/Shapes/Geometry3D/Functions/GetLinkingLine3D

	{attribute 'TcIecLibraryType'}
	{attribute 'external_name' := 'GetLinkingLine3D_GUID_571B8048_3BB2_3575_4227_68A764324927'}
	(* Get the shortest path between two geometries. *)
	FUNCTION GetLinkingLine3D : BOOL
	VAR_IN_OUT
		geometry0	:	IPlcGeometry3D;	(* 1st input geometry to calculate the linking line for. *)
		geometry1	:	IPlcGeometry3D;	(* 2nd input geometry to calculate the linking line for. *)
		linkingLine	:	Segment3D;	(* Return the resulting linking line. *)
	END_VAR

END_FUNCTION

// POUs/Shapes/Geometry3D/Functions/CreateIntersection2D

	{attribute 'TcIecLibraryType'}
	{attribute 'external_name' := 'CreateIntersection2D_GUID_6BC618A5_CC8E_3E0D_5D09_850F7B7B2EA3'}
	(* Create a collection of intersections along a plane definition. *)
	FUNCTION CreateIntersection2D : BOOL
	VAR_IN_OUT
		container3D	:	Container3D;	(* Input container to create the intersections of. *)
		planeFrame	:	PositionSE3;	(* The coordinate frame to indicate the origin of the plane. *)
		container2D	:	Container2D;	(* Return the resulting collection of intersection. *)
	END_VAR

END_FUNCTION
